FUNCTION_BLOCK MQTT_3 (* Peroidic event generator *)
  (* Standard: 61499-1 Annex A; Description: Copyright (c) 2017 fortiss GmbH This program and the accompanying materials are made available under the terms of the Eclipse Public License 2.0 which is available at https://www.eclipse.org/legal/epl-2.0/ SPDX-License-Identifier: EPL-2.0 *)
  (* Version 1.0, 2017-09-21, Alois Zoitl, fortiss GmbH, initial API and implementation and/or initial documentation *)
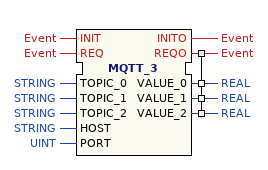
  EVENT_INPUT
    INIT;
    REQ;
  END_EVENT
  EVENT_OUTPUT
    INITO;
    REQO WITH VALUE_0, VALUE_1, VALUE_2;
  END_EVENT
  VAR_INPUT
    TOPIC_0 : STRING;
    TOPIC_1 : STRING;
    TOPIC_2 : STRING;
    HOST : STRING;
    PORT : UINT;
  END_VAR
  VAR_OUTPUT
    VALUE_0 : REAL;
    VALUE_1 : REAL;
    VALUE_2 : REAL;
  END_VAR
END_FUNCTION_BLOCK
